// TIA Portal V21 export
TYPE "LBC_typeAnalogOutputInterface"
TITLE = LBC_typeAnalogOutputInterface
// Module interface for external systems
   STRUCT
      commands : "LBC_typeInterfaceCommands";
      monitoring { ExternalWritable := 'False'} : "LBC_typeAnalogProcessValues";
      configuration : "LBC_typeAnalogOutputConfiguration";
   END_STRUCT;
END_TYPE
